PROGRAM PRG_MasterSystemTime
VAR
	//Variables
	bReadyToRead				:BOOL;
	bFirstScan					:BOOL := TRUE;
	bUpdateSysTime				:BOOL; //Output of pulse generator
	tSysTimeUpdatePeriod		:TIME := T#5S;
	stTimeStamp					:TIMESTRUCT;
	stNullTimeStamp				:TIMESTRUCT;
	sRawDateTime				:STRING;
	sSystemDate					:STRING;
	sSystemTime					:STRING;
	sDateTime					:STRING;
	sDateTimeSpaces				:STRING;
	
	stTimeTest                  :TIMESTRUCT;
	sttimeTest2                 :TIMESTRUCT;
	sTestTime                   :STRING;
	nSectTest                   :DINT;
	bStartTest                  :BOOL;
	bStsrtTest2                 :BOOL;
	
	
	//Functions
	fbGetSystemTime				:TC2_Utilities.NT_GetTime;
	fbRTClock					:TC2_Utilities.RTC_EX2;		//Local real-time clock
	tonTimeUpdateGen			:TC2_Utilities.TON;			//Pulse generator for triggering fbGetSystemTime function
	rtrigSysTimeCollected		:TC2_Utilities.R_TRIG;		//System time collected

    fbTimerControl              :FB_TimeControl;
	bStartTimeTest              :BOOL;
	bResetTimeTest              :BOOL;
	nTimeHourTest               :DINT;
	nTimeMinTest                :DINT;
	nTimeSecTest                :DINT;
	nTimeTotalSecTest           :DINT;
END_VAR

//Aux functions call
tonTimeUpdateGen(	IN := NOT bUpdateSysTime,
					PT := tSysTimeUpdatePeriod,
					Q => bUpdateSysTime);

//bReadyToRead :=  Tc2_System.MEMCMP( ADR( stTimeStamp), ADR (stNullTimeStamp), SIZEOF(stTimeStamp)) <> 0 AND NOT  fbGetSystemTime.BUSY;	
			(*keczi*)	(*zrobione po to zeby w wypadku jak po starcie PLC na HMI mial pokazywac czas alarmu '00:00:00', zebyb poczekal az faktycznie pokazuje date i czas*)

//Get Current System Time
fbGetSystemTime(NETID := ,
				START := bFirstScan OR bUpdateSysTime,
				TMOUT := ,
				BUSY => ,
				ERR => ,
				ERRID => ,
				TIMESTR => );
				
//Get system time done detection - one-shot
rtrigSysTimeCollected(CLK := NOT fbGetSystemTime.BUSY);

//Synchronize Real-Time clock with system time
fbRTClock(	EN := rtrigSysTimeCollected.Q, 
			PDT := fbGetSystemTime.TIMESTR,
			CDT => stTimeStamp, 
			Q => bReadyToRead);

// System Date and Time in Proper Order 
IF bReadyToRead THEN
	sRawDateTime := SYSTEMTIME_TO_STRING(stTimeStamp);  // format: YYYY-MM-DD-hh:mm:ss.xxx
	sSystemDate := CONCAT(CONCAT(CONCAT(CONCAT(MID(sRawDateTime, 2, 9), '.'),  MID(sRawDateTime, 2, 6)), '.'), LEFT(sRawDateTime, 4));
	sSystemTime := MID(sRawDateTime, 8, 12);
	sDateTime := CONCAT(CONCAT(sSystemDate, '  '), sSystemTime);
	sDateTimeSpaces	:= CONCAT(sDateTime, '    ');
	
	//Time to write to CSV Files
	//nSystemTime := sSystemTime;
END_IF;

bFirstScan := FALSE;

IF bStartTest THEN
	sTestTime:= SYSTEMTIME_TO_STRING(stTimeTest);
END_IF

fbTimerControl( bEnable  :=  bStartTimeTest,
	            bReset   :=  bResetTimeTest,
				nHour     => nTimeHourTest,
				nMin      => nTimeMinTest,
				nSec      => nTimeSecTest,
				nTotalSec => nTimeTotalSecTest );

END_PROGRAM

(* stored: Version 1.1.0.1, ProductVersion 3.1.4024.13
   POU PRG_MasterSystemTime: Id {7173042a-7f7f-45b8-b04e-de7c8939b16f}, SpecialFunc None *)
